(* IEC 61131-3 sources: AXOpen/src/components.festo.drives/ctrl/src (part 3) *)

(* ---- AxoCmmtAsPtP_PositioningIn.st ---- *)
NAMESPACE AXOpen.Components.Festo.Drives
    {S7.extern=ReadWrite}
    CLASS AxoCmmtAsPtP_PositioningIn
        VAR PUBLIC
            {#ix-attr:[Container(Layout.Stack)]}
            {#ix-set:AttributeName = "<#ModePos#>"}
            ModePos				:	INT		:=	INT#2;
            {#ix-set:AttributeName = "<#EnableAxis#>"}
            EnableAxis			:	BOOL	:=	FALSE;
            {#ix-set:AttributeName = "<#CancelTraversing#>"}
            CancelTraversing	:	BOOL	:=	TRUE;
            {#ix-set:AttributeName = "<#IntermediateStop#>"}
            IntermediateStop	:	BOOL	:=	TRUE;
            {#ix-set:AttributeName = "<#Positive#>"}
            Positive			:	BOOL	:=	FALSE;
            {#ix-set:AttributeName = "<#Negative#>"}
            Negative			:	BOOL	:=	FALSE;
            {#ix-set:AttributeName = "<#Jog1#>"}
            Jog1				:	BOOL	:=	FALSE;
            {#ix-set:AttributeName = "<#Jog2#>"}
            Jog2				:	BOOL	:=	FALSE;
            {#ix-set:AttributeName = "<#AckError#>"}
            AckError			:	BOOL	:=	FALSE;
            {#ix-set:AttributeName = "<#ExecuteMode#>"}
            ExecuteMode			:	BOOL	:=	FALSE;
            {#ix-set:AttributeName = "<#ReleaseBrake#>"}
            ReleaseBrake		:	BOOL	:=	FALSE;
            {#ix-set:AttributeName = "<#TravelToFixStop#>"}
            TravelToFixStop		:	BOOL	:=	FALSE;
            {#ix-set:AttributeName = "<#Position#>"}
            Position			:	DINT	:=	DINT#0;
            {#ix-set:AttributeName = "<#Velocity#>"}
            Velocity			:	DINT	:=	DINT#0;
            {#ix-set:AttributeName = "<#OverV#>"}
            OverV				:	INT		:=	INT#100;
            {#ix-set:AttributeName = "<#OverAcc#>"}
            OverAcc				:	INT		:=	INT#100;
            {#ix-set:AttributeName = "<#OverDec#>"}
            OverDec				:	INT		:=	INT#100;
            {#ix-set:AttributeName = "<#ConfigEPos#>"}
            ConfigEPos			:	DWORD	:=	DWORD#16#0000_000F;
            {#ix-set:AttributeName = "<#BaseSpeedValue#>"}
            BaseSpeedValue		:	REAL	:=	REAL#0.0;
            {#ix-set:AttributeName = "<#AdditionalTorque#>"}
            AdditionalTorque	:	REAL	:=	REAL#0.0;
            {#ix-set:AttributeName = "<#PositiveTorqueLimit#>"}
            PositiveTorqueLimit	:	REAL	:=	REAL#100.0;
            {#ix-set:AttributeName = "<#NegativeTorqueLimit#>"}
            NegativeTorqueLimit	:	REAL	:=	REAL#100.0;
        END_VAR
    END_CLASS
END_NAMESPACE

(* ---- AxoCmmtAsPtPAxisData.st ---- *)
NAMESPACE AXOpen.Components.Festo.Drives
    {S7.extern=ReadWrite}
    CLASS AxoCmmtAsPtPAxisData
        VAR PUBLIC
            MAP_HW_ID   :   ULINT;
        END_VAR
    END_CLASS
END_NAMESPACE

(* ---- AxoCmmtAsPtPAxisReference.st ---- *)
// USING AXOpen.Components.Drives;

NAMESPACE AXOpen.Components.Festo.Drives
    {S7.extern=ReadWrite}
    CLASS AxoCmmtAsPtPAxisReference
        VAR PUBLIC
            Telegram111_In      :   AXOpen.Components.Festo.Drives.PROFIdriveTelegram_111_IN;
            Telegram111_Out     :   AXOpen.Components.Festo.Drives.PROFIdriveTelegram_111_OUT;
            Telegram750_In      :   AXOpen.Components.Festo.Drives.PROFIdriveTelegram_750_IN;
            Telegram750_Out     :   AXOpen.Components.Festo.Drives.PROFIdriveTelegram_750_OUT;
            Data                :   AXOpen.Components.Festo.Drives.AxoCmmtAsPtPAxisData;
            Config              :   AXOpen.Components.Drives.AxoDrive_Config;
            Status              :   AXOpen.Components.Drives.AxoDrive_Status;
        END_VAR
    END_CLASS
END_NAMESPACE

(* ---- AxoPROFIdriveParametrizationIn.st ---- *)
USING AXOpen.Core;
USING Siemens.Simatic.S71500.DistributedIO;

NAMESPACE AXOpen.Components.Festo.Drives
    {S7.extern=ReadWrite}
    CLASS AxoPROFIdriveParametrizationIn
        VAR PUBLIC
            {#ix-attr:[Container(Layout.Stack)]}
            {#ix-set:AttributeName = "<#Enable#>"}
            Enable          :   BOOL;
            {#ix-set:AttributeName = "<#ReadWrite#>"}
            ReadWrite       :   BOOL;
            {#ix-set:AttributeName = "<#ParameterNo#>"}
            ParameterNo     :   INT;
            {#ix-set:AttributeName = "<#Subindex#>"}
            Subindex        :   INT;
            {#ix-set:AttributeName = "<#AxisNo#>"}
            AxisNo	        :   BYTE := BYTE#1;
            {#ix-set:AttributeName = "<#HardwareId#>"}
            HardwareId	    :   WORD;
            {#ix-set:AttributeName = "<#ValueWriteREAL#>"}
            ValueWriteREAL  :   REAL;
            {#ix-set:AttributeName = "<#ValueWriteLINT#>"}
            ValueWriteLINT  :   LINT;
            {#ix-set:AttributeName = "<#ValueWriteBOOL#>"}
            ValueWriteBOOL  :   BOOL;
        END_VAR
    END_CLASS
END_NAMESPACE

(* ---- AxoReadWritePROFIdriveParameter.st ---- *)
USING AXOpen.Core;
USING Siemens.Simatic.S71500.DistributedIO;

NAMESPACE AXOpen.Components.Festo.Drives
    {S7.extern=ReadWrite}
    CLASS AxoReadWritePROFIdriveParameter EXTENDS AXOpen.Core.AxoObject
        VAR PUBLIC
            Enable          :   BOOL;
            ReadWrite       :   BOOL;
            ParameterNo     :   INT;
            Subindex        :   INT;
            AxisNo	        :   BYTE;
            HardwareId	    :   WORD;
        END_VAR

        VAR PUBLIC
            ValueReadREAL  :   REAL;
            ValueReadLINT  :   LINT;
            ValueReadBOOL  :   BOOL;
        END_VAR

        VAR PUBLIC
            ValueWriteREAL  :   REAL;
            ValueWriteLINT  :   LINT;
            ValueWriteBOOL  :   BOOL;
        END_VAR

        VAR PUBLIC
            Busy	:   BOOL;
            Done	:   BOOL;
            Error	:   BOOL;
            ErrorId :	DWORD;
        END_VAR

        VAR PRIVATE
            Enable_PV   :   BOOL;

            Busy_	:   BOOL;
            Done_	:   BOOL;
            Error_	:   BOOL;
            ErrorId_:	DWORD;
            StartTimer : BOOL;
            StartRW : BOOL;

            AxoOnDelatTimer :  AXOpen.Timers.OnDelayTimer;

            RW_Data         :   ARRAY[0..9] OF BYTE;
            WR_Data         :   ARRAY[0..19] OF BYTE;
            RD_Data         :   ARRAY[0..13] OF BYTE;
            RW_Status        :	DWORD;
            WR_Status        :	DWORD;
            RD_Status        :	DWORD;

            ReadRecord_     :   ReadRecord;
            WriteRecord_    :   WriteRecord;
            ErrorCounter    :	UINT;

            LengthRead      :	UINT;
            State           :   INT;
            ReqRef          :   BYTE;
            wordhlp         :   WORD;
        END_VAR

        VAR CONSTANT PRIVATE
            LenHeader	    :   UINT    :=	UINT#4;
            LenRequest	    :   UINT    :=  UINT#6;
            LenWrite	    :   UINT    :=  UINT#16;
            LenRead	        :   UINT    :=  UINT#10;
            PD_Error	    :   DWORD	:=  DWORD#16#4000_0000;
            MaxRetryCounter	:   UINT    :=	UINT#150;

        END_VAR

        METHOD PUBLIC Run
            VAR_INPUT
                parent          :   IAxoObject;
            END_VAR

            THIS.Initialize(parent);
            THIS.Execute();

        END_METHOD

        METHOD PUBLIC Run
            VAR_INPUT
                parent          :   IAxoContext;
            END_VAR

            THIS.Initialize(parent);
            THIS.Execute();

        END_METHOD

        METHOD PUBLIC Execute

            VAR
                _lenght     :   UINT;
                i           :   INT;
                tmpWord     :   WORD;
                tmpSINT     :   SINT;
                tmpINT      :   INT;
                tmpDINT     :   DINT;
                tmpDWORD    :   DWORD;
                tmpLINT     :   LINT;
            END_VAR

                //Check the Inputs
                IF HardwareId = WORD#0 THEN
                    Error_ := TRUE;
                    ErrorId_ := DWORD#16#00001010;    //HardwareID = 0
                    RETURN;
                END_IF;

                //Timer
                AxoOnDelatTimer.OnDelay(THIS, StartTimer,T#100MS);

                IF AxoOnDelatTimer.output THEN
                    StartRW := TRUE;
                    StartTimer := FALSE;
                END_IF;

                IF State = 0 THEN //Wait for start trigger
                    IF Enable AND NOT Enable_PV THEN
                        StartRW := TRUE;
                        State := 10;
                        Busy := TRUE;
                    END_IF;
                END_IF;

                IF State = 10 THEN
                    (* ------------------ HEADER --------------------*)
                    //Request reference starts with 1 and will count up
                    RW_Data[0] := ReqRef;
                    // Requst ID = 1 (Request Parameter)
                    RW_Data[1] := BYTE#1;
                    //Fill the Axis number
                    RW_Data[2] := AxisNo;
                    // Single parameter access
                    RW_Data[3] := BYTE#1;
                    (* ------------------ Parameter address ------------*)
                    //Attribute
                    RW_Data[4]:= BYTE#16#10;
                    //ElemNo.
                    RW_Data[5] := BYTE#1;
                    // Assign PNU
                    RW_Data[6] := ParameterNo.%B1;
                    RW_Data[7] := ParameterNo.%B0;
                    // Assign Subindex
                    RW_Data[8] := Subindex.%B1;
                    RW_Data[9] := Subindex.%B0;

                    // Lenght of the telegramm to be send
                    _lenght := LenHeader + LenRequest;

                    WriteRecord_(request    :=  StartRW,
                                id          :=  HardwareId,
                                index       :=  16#b02e,
                                length      :=  _lenght,
                                record      :=  RW_Data,
                                status      =>  WR_Status);

                    IF WriteRecord_.DONE THEN
                        ErrorCounter := UINT#0;
                        //delete old response values
                        FOR i := 0 TO 13 DO
                            RD_Data[i] := BYTE#0;
                        END_FOR;

                        IF NOT ReadWrite THEN
                            //Read parameter
                            State := 20;
                        ELSE
                            //Write parameter
                            State := 50;
                        END_IF;
                    ELSIF WriteRecord_.ERROR THEN
                        tmpWord := TO_WORD(TO_DINT(WR_Status)/256);
                        wordhlp := tmpWord;
                        //try it again
                        IF ((tmpWord = WORD#16#80A7) OR (tmpWord = WORD#16#80B5) OR (tmpWord = WORD#16#80C0) OR (tmpWord = WORD#16#80C1) OR (tmpWord = WORD#16#80C2)
                            OR (tmpWord = WORD#16#80C3) OR (tmpWord = WORD#16#80C4)) AND (ErrorCounter < MaxRetryCounter) THEN
                            ErrorCounter := ErrorCounter + UINT#1;
                            StartRW := FALSE;
                            StartTimer := TRUE;
                        ELSE
                            State := 70;
                        END_IF;

                    END_IF;
                END_IF;

                IF State = 20 THEN  //Read Parameter
                    // Lenght of the telegramm for reading
                    _lenght := LenHeader + LenRead;

                    ReadRecord_(request     :=  StartRW,
                                id          :=  HardwareId,
                                index       :=  16#b02e,
                                maxLength   :=  _lenght,
                                record      :=  RD_Data,
                                status      =>  RD_Status,
                                length      =>  LengthRead);

                    IF ReadRecord_.VALID AND NOT ReadRecord_.BUSY THEN
                        ErrorCounter := UINT#0;
                        State := 30;
                    ELSIF ReadRecord_.ERROR THEN
                        tmpWord := TO_WORD(TO_DINT(RD_Status) / 256);
                        wordhlp := tmpWord;
                        //try it again
                        IF ((tmpWord = WORD#16#80A7) OR (tmpWord = WORD#16#80B5) OR (tmpWord = WORD#16#80C0) OR (tmpWord = WORD#16#80C1) OR (tmpWord = WORD#16#80C2)
                            OR (tmpWord = WORD#16#80C3) OR (tmpWord = WORD#16#80C4)) AND (ErrorCounter < MaxRetryCounter) THEN
                            ErrorCounter := ErrorCounter + UINT#1;
                            StartRW := FALSE;
                            StartTimer := TRUE;
                        ELSE
                            State := 80;
                        END_IF;
                    END_IF;
                END_IF;

                IF State = 30 THEN //Reading finished successfull

                    CASE TO_INT(RD_Data[4]) OF //Format
                        0:  //reserved
                            ValueReadREAL := REAL#0.0;
                            ValueReadLINT := LINT#0;
                            ValueReadBOOL := FALSE;

                            ErrorId := DWORD#16#1001;    //reserved DataType
                            // #Error
                            State := 200;

                        1:  // BOOLEAN
                            //copy the value to the output
                            ValueReadREAL := 0;
                            ValueReadLINT := 0;
                            ValueReadBOOL := TO_BOOL(RD_Data[6]);

                            // no error
                            State := 100;

                        2:  //SINT8
                            tmpSINT := TO_SINT(RD_Data[6]);
                            //copy the value to the output
                            ValueReadREAL := 0;
                            ValueReadLINT := (TO_LINT(tmpSINT));
                            ValueReadBOOL := FALSE;

                            // no error
                            State := 100;

                        3:  //SINT16
                            tmpINT.%B0 := RD_Data[7];
                            tmpINT.%B1 := RD_Data[6];

                            //copy the value to the output
                            ValueReadREAL := 0;
                            ValueReadLINT := TO_LINT(tmpINT);
                            ValueReadBOOL := FALSE;

                            // no #Error
                            State := 100;

                        4:  //SINT32
                            tmpDINT.%B0 := RD_Data[9];
                            tmpDINT.%B1 := RD_Data[8];
                            tmpDINT.%B2 := RD_Data[7];
                            tmpDINT.%B3 := RD_Data[6];

                            //copy the value to the output
                            ValueReadREAL := 0;
                            ValueReadLINT := TO_LINT(tmpDINT);
                            ValueReadBOOL := FALSE;

                            // no #Error
                            State := 100;

                        5, 65: //USINT8(5) or BYTE(65)
                            //copy the value to the output
                            ValueReadREAL := 0;
                            ValueReadLINT := (TO_LINT(RD_Data[6]));
                            ValueReadBOOL := FALSE;

                            // no error
                            State := 100;

                        6, 66: //UINT16(6) or WORD(66)
                            tmpWord.%B0 := RD_Data[7];
                            tmpWord.%B1 := RD_Data[6];

                            //copy the value to the output
                            ValueReadREAL := 0;
                            ValueReadLINT := TO_LINT(tmpWord);
                            ValueReadBOOL := FALSE;

                            // no #Error
                            State := 100;

                        7, 67: //UDINT32(7) or DWORD(67)
                            tmpDWord.%B0 := RD_Data[9];
                            tmpDWord.%B1 := RD_Data[8];
                            tmpDWord.%B2 := RD_Data[7];
                            tmpDWord.%B3 := RD_Data[6];

                            //copy the value to the output
                            ValueReadREAL := 0;
                            ValueReadLINT := TO_LINT(tmpDWord);
                            ValueReadBOOL := FALSE;

                            // no #Error
                            State := 100;

                        8:  //FLOAT32
                            tmpDWord.%B0 := RD_Data[9];
                            tmpDWord.%B1 := RD_Data[8];
                            tmpDWord.%B2 := RD_Data[7];
                            tmpDWord.%B3 := RD_Data[6];

                            //copy the value to the output
                            ValueReadREAL := TO_REAL(tmpDWord);
                            ValueReadLINT := 0;
                            ValueReadBOOL := FALSE;

                            // no #Error
                            State := 100;

                        10:  //OctetString
                            tmpINT.%B0 := RD_Data[6];
                            tmpINT.%B1 := RD_Data[7];

                            //copy the value to the output
                            ValueReadREAL := 0;
                            ValueReadLINT := TO_LINT(tmpINT);
                            ValueReadBOOL := FALSE;

                            // no #Error
                            State := 100;

                        55, 56:  //LINT, ULINT
                            tmpLINT.%B0 :=RD_Data[13];
                            tmpLINT.%B1 :=RD_Data[12];
                            tmpLINT.%B2 :=RD_Data[11];
                            tmpLINT.%B3 :=RD_Data[10];
                            tmpLINT.%B4 :=RD_Data[9];
                            tmpLINT.%B5 :=RD_Data[8];
                            tmpLINT.%B6 :=RD_Data[7];
                            tmpLINT.%B7 :=RD_Data[6];

                            //copy the value to the output
                            ValueReadREAL := 0;
                            ValueReadLINT := tmpLINT;
                            ValueReadBOOL := FALSE;

                            // no #Error
                            State := 100;

                        68:  //Error
                            tmpDWord.%B0 := RD_Data[7];
                            tmpDWord.%B1 := RD_Data[6];
                            ErrorId := tmpDWord OR PD_Error;

                            //copy the value to the output
                            ValueReadREAL := 0;
                            ValueReadLINT := 0;
                            ValueReadBOOL := FALSE;

                            // #Error
                            State := 200;

                        ELSE
                            ValueReadREAL := 0;
                            ValueReadLINT := 0;
                            ValueReadBOOL := FALSE;

                            ErrorId := DWORD#16#1000;    //unknown DataType
                            // #Error
                            State := 200;
                    END_CASE;
                END_IF;

                IF State = 50 THEN //Write Parameter (First Read dataset then write dataset)
                    // Lenght of the telegramm for reading
                    _lenght := LenHeader + LenRead;

                    ReadRecord_(request     :=  StartRW,
                                id          :=  HardwareId,
                                index       :=  16#b02e,
                                maxLength   :=  _lenght,
                                record      :=  RD_Data,
                                status      =>  RD_Status,
                                length      =>  LengthRead);

                    IF ReadRecord_.VALID AND NOT ReadRecord_.BUSY THEN
                        ErrorCounter := UINT#0;
                        State := 55;
                    ELSIF ReadRecord_.ERROR THEN
                        tmpWord := TO_WORD(TO_DINT(RD_Status)/256);
                        wordhlp := tmpWord;
                        //try it again
                        IF ((tmpWord = WORD#16#80A7) OR (tmpWord = WORD#16#80B5) OR (tmpWord = WORD#16#80C0) OR (tmpWord = WORD#16#80C1) OR (tmpWord = WORD#16#80C2)
                            OR (tmpWord = WORD#16#80C3) OR (tmpWord = WORD#16#80C4)) AND (ErrorCounter < MaxRetryCounter) THEN
                            ErrorCounter := ErrorCounter + UINT#1;
                            StartRW := false;
                            StartTimer := TRUE;
                        ELSE
                            State := 80;
                        END_IF;
                    END_IF;
                END_IF;

                IF State = 55 THEN //Reading finished
                    CASE TO_INT(RD_Data[4]) OF // Format
                        0:  //reserved
                            ValueReadREAL := 0;
                            ValueReadLINT := 0;
                            ValueReadBOOL := FALSE;

                            ErrorId := DWORD#16#1001;    //reserved DataType
                            // #Error
                            State := 200;

                        1, 2, 3, 4, 5, 6, 7, 8, 55, 56, 65, 66, 67:
                            State := 60;

                        68:  //Error
                            tmpDWord.%B0 := RD_Data[7];
                            tmpDWord.%B1 := RD_Data[6];
                            ErrorId := tmpDWord OR PD_Error;

                            //copy the value to the output
                            ValueReadREAL := 0;
                            ValueReadLINT := 0;
                            ValueReadBOOL := FALSE;

                            // #Error
                            State := 200;

                        ELSE
                            ValueReadREAL := 0;
                            ValueReadLINT := 0;
                            ValueReadBOOL := FALSE;

                            ErrorId := DWORD#16#1000;    //unknown DataType
                            // #Error
                            State := 200;
                    END_CASE;
                END_IF;

                IF State = 60 THEN //reading Done from Write request
                    (* ------------------ HEADER --------------------*)
                    //Request reference starts with 1 and will count up
                    WR_Data[0] := TO_BYTE(TO_INT(ReqRef) + 1);
                    // Requst ID = 2 (Change Parameter)
                    WR_Data[1] := BYTE#2;
                    //Fill the Axis number
                    WR_Data[2] := AxisNo;
                    // Single parameter access
                    WR_Data[3] := BYTE#1;
                    (* ------------------ DATA --------------------*)
                    // Attribute
                    WR_Data[4] := BYTE#16#10;
                    // Single Access
                    WR_Data[5] := BYTE#1;
                    // PNU
                    WR_Data[6] := ParameterNo.%B1;
                    WR_Data[7] := ParameterNo.%B0;
                    // Subindex
                    WR_Data[8] := Subindex.%B1;
                    WR_Data[9] := Subindex.%B0;
                    //Format
                    WR_Data[10] := RD_Data[4];
                    //No. Values
                    WR_Data[11] := BYTE#1;
                    //erase send buffer
                    FOR i := 12 TO 19 DO
                        WR_Data[i] := BYTE#0;
                    END_FOR;

                    CASE TO_INT(RD_Data[4]) OF //Format
                        0:  //reserved
                            ValueReadREAL := 0;
                            ValueReadLINT := 0;
                            ValueReadBOOL := FALSE;

                            ErrorId := DWORD#16#1001;    //reserved DataType
                            // #Error
                            State := 200;

                        1:  //BOOL
                            WR_Data[12] := TO_BYTE(ValueWriteBOOL);

                        2, 5, 65:  //SINT8, USINT8, BYTE
                            WR_Data[12] := TO_BYTE(ValueWriteLINT);

                        3, 6, 66:  //SINT16, UINT16, WORD
                            WR_Data[12] := ValueWriteLINT.%B1;
                            WR_Data[13] := ValueWriteLINT.%B0;

                        4, 7, 67: //SINT32, UDINT32, DWORD
                            WR_Data[12] := ValueWriteLINT.%B3;
                            WR_Data[13] := ValueWriteLINT.%B2;
                            WR_Data[14] := ValueWriteLINT.%B1;
                            WR_Data[15] := ValueWriteLINT.%B0;

                        8:  //FLOAT32
                            tmpDWORD    :=  TO_DWORD(ValueWriteREAL);
                            WR_Data[12] := tmpDWORD.%B3;
                            WR_Data[13] := tmpDWORD.%B2;
                            WR_Data[14] := tmpDWORD.%B1;
                            WR_Data[15] := tmpDWORD.%B0;

                        55, 56:  //SINT64
                            WR_Data[12] := ValueWriteLINT.%B7;
                            WR_Data[13] := ValueWriteLINT.%B6;
                            WR_Data[14] := ValueWriteLINT.%B5;
                            WR_Data[15] := ValueWriteLINT.%B4;
                            WR_Data[16] := ValueWriteLINT.%B3;
                            WR_Data[17] := ValueWriteLINT.%B2;
                            WR_Data[18] := ValueWriteLINT.%B1;
                            WR_Data[19] := ValueWriteLINT.%B0;

                    END_CASE;

                    //goto the next step
                    State := 61;
                END_IF;

                IF State = 61 THEN //send the write Request
                    // Lenght of the telegramm to be send
                    _lenght := LenHeader + LenWrite;

                    WriteRecord_(request    :=  StartRW,
                                id          :=  HardwareId,
                                index       :=  16#b02e,
                                length      :=  _lenght,
                                record      :=  WR_Data,
                                status      =>  RW_Status);

                    IF WriteRecord_.DONE THEN
                        State := 62;
                    ELSIF WriteRecord_.ERROR THEN
                        tmpWord := TO_WORD(TO_DINT(RW_Status)/256);
                        wordhlp := tmpWord;
                        //try it again
                        IF ((tmpWord = WORD#16#80A7) OR (tmpWord = WORD#16#80B5) OR (tmpWord = WORD#16#80C0) OR (tmpWord = WORD#16#80C1) OR (tmpWord = WORD#16#80C2)
                            OR (tmpWord = WORD#16#80C3) OR (tmpWord = WORD#16#80C4)) AND (ErrorCounter < MaxRetryCounter) THEN
                            ErrorCounter := ErrorCounter + UINT#1;
                            StartRW := FALSE;
                            StartTimer := TRUE;
                        ELSE
                            State := 90;
                        END_IF;
                    END_IF;
                END_IF;

                IF State = 62 THEN //Read the answer of the write request

                    //delete old response values
                    FOR i := 0 TO 13 DO
                        RD_Data[i] := BYTE#0;
                    END_FOR;

                    // Lenght of the telegramm for reading
                    _lenght := LenHeader + LenRead;

                    ReadRecord_(request     :=  StartRW,
                                id          :=  HardwareId,
                                index       :=  16#b02e,
                                maxLength   :=  _lenght,
                                record      :=  RD_Data,
                                status      =>  RD_Status,
                                length      =>  LengthRead);

                    IF ReadRecord_.VALID AND NOT ReadRecord_.BUSY THEN
                        ErrorCounter := UINT#0;
                        State := 63;
                    ELSIF ReadRecord_.ERROR THEN
                        tmpWord := TO_WORD(TO_DINT(RD_Status)/256);
                        wordhlp := tmpWord;
                        //try it again
                        IF ((tmpWord = WORD#16#80A7) OR (tmpWord = WORD#16#80B5) OR (tmpWord = WORD#16#80C0) OR (tmpWord = WORD#16#80C1) OR (tmpWord = WORD#16#80C2)
                            OR (tmpWord = WORD#16#80C3) OR (tmpWord = WORD#16#80C4)) AND (ErrorCounter < MaxRetryCounter) THEN
                            ErrorCounter := ErrorCounter + UINT#1;
                            StartRW := FALSE;
                            StartTimer := TRUE;
                        ELSE
                            State := 80;
                        END_IF;
                    END_IF;
                END_IF;

                IF State = 63 THEN //Reading finished

                    CASE TO_INT(RD_Data[1]) OF //ReqId

                        2:  //positive resonse
                            State := 150;

                        128..130:  //negative response
                            IF RD_Data[4] = BYTE#68 THEN //Format
                                tmpDWord.%B0 := RD_Data[7];
                                tmpDWord.%B1 := RD_Data[6];
                                ErrorId := tmpDWord OR PD_Error;

                                // #Error
                                State := 200;
                            ELSE
                                ErrorId := DWORD#16#1003; //negative response without error code
                                State := 300;
                            END_IF;
                        ELSE  //undefined response ID
                            ErrorId := DWORD#16#1002;
                            State := 300;
                    END_CASE;
                END_IF;

                IF State = 70 THEN // Error while ReadWrite Access
                    Done := TRUE;
                    Busy := FALSE;
                    Error := TRUE;
                    ErrorId := WR_Status;
                END_IF;

                IF State = 80 THEN //Error Reading Access
                    Done := TRUE;
                    Busy := FALSE;
                    Error := TRUE;
                    ErrorId := RD_Status;
                END_IF;

                IF State = 90 THEN // Error while Write Access
                    Done := TRUE;
                    Busy := FALSE;
                    Error := TRUE;
                    ErrorId := RW_Status;
                END_IF;

                IF State = 100 THEN // read successfully
                    Done := TRUE;
                    Busy := FALSE;
                    Error := FALSE;
                END_IF;

                IF State = 150 THEN // write successfully
                    Done := TRUE;
                    Busy := FALSE;
                    Error := FALSE;
                END_IF;

                IF State = 200 THEN //Error while reading
                    Done := TRUE;
                    Busy := FALSE;
                    Error := TRUE;

                    IF State = 300 THEN //Error while writing
                        Done := TRUE;
                        Busy := FALSE;
                        Error := TRUE;
                    END_IF;
                END_IF;

                IF NOT Enable THEN
                    State := 0;
                    ReqRef := BYTE#1;
                    Done := FALSE;
                    Busy := FALSE;
                    Error := FALSE;
                    ErrorId := DWORD#16#00000000;
                    ValueReadBOOL := FALSE;
                    ValueReadLINT := 0;
                    ValueReadREAL := 0;
                    RD_Status := DWORD#0;
                    ErrorCounter := UINT#0;
                END_IF;

                Enable_PV := Enable;

        END_METHOD
    END_CLASS
END_NAMESPACE
